PROGRAM MAIN
VAR
	bFirstCycle		: BOOL := TRUE;
END_VAR



P02_GlobalSystemTime();
P03_MachineControl();
P03_MachineControl.Robot();
P03_MachineControl.Batch();
P05_DeviceControl();
P06_ProcessControl();
P99_HMIControl();

//Simulations
Service_sim();



bFirstCycle := FALSE;

END_PROGRAM

(* stored: Version 1.1.0.1
   POU MAIN: Id {b327c351-3beb-4a3c-9556-c753d3115e3b}, SpecialFunc None *)
